// TIA Portal V15.1 export
// export: Created 2024-05-17T05:38:17.1171351Z, ExportSetting WithDefaults, DisplayName Totally Integrated Automation Portal, DisplayVersion V15.1 Update 5, DisplayName TIA Portal Openness, DisplayVersion V15.1 Update 5, DisplayName SINAMICS Startdrive Advanced, DisplayVersion V15.1, DisplayName G130, G150, S120, S150, SINAMICS MV, S210, DisplayVersion V15.1, DisplayName G110M, G120, G120C, G120D, G120P, DisplayVersion V15.1, DisplayName STEP 7 Professional, DisplayVersion V15.1 Update 5, DisplayName STEP 7 Safety, DisplayVersion V15.1, DisplayName WinCC Professional, DisplayVersion V15.1 Update 5, DisplayName SIMATIC Visualization Architect, DisplayVersion V15.1
DATA_BLOCK "_209220ZS01Passiv"   // DB373
{ S7_Optimized_Access := 'FALSE' }
AUTHOR : VCC
VERSION : 0.1
// stored: AutoNumber false, DBAccessibleFromOPCUA true, IsOnlyStoredInLoadMemory false, IsWriteProtectedInAS false
   VAR RETAIN
      AA_209000AK04JX37QF5270 { ExternalAccessible := 'False'; ExternalVisible := 'False'; ExternalWritable := 'False'} : Bool;   // Passivation alarm - ET200sp I/O - Safety Card QF5270
      AA_209000AK04JX37QF5276 { ExternalAccessible := 'False'; ExternalVisible := 'False'; ExternalWritable := 'False'} : Bool;   // Passivation alarm - ET200sp I/O - Safety Card QF5276
      AA_209220AS10JX50IF6000 { ExternalAccessible := 'False'; ExternalVisible := 'False'; ExternalWritable := 'False'} : Bool;   // Passivation alarm - ET200sp I/O - Safety Card IF6000
      AA_209220AX01JX51IF6050 { ExternalAccessible := 'False'; ExternalVisible := 'False'; ExternalWritable := 'False'} : Bool;   // Passivation alarm - ET200sp I/O - Safety Card IF6050
      AA_209220AS11JX52IF6100 { ExternalAccessible := 'False'; ExternalVisible := 'False'; ExternalWritable := 'False'} : Bool;   // Passivation alarm - ET200sp I/O - Safety Card IF6100
      AA_209220AX02JX53IF6150 { ExternalAccessible := 'False'; ExternalVisible := 'False'; ExternalWritable := 'False'} : Bool;   // Passivation alarm - ET200sp I/O - Safety Card IF6150
      AA_209220AS20JX58IF6200 { ExternalAccessible := 'False'; ExternalVisible := 'False'; ExternalWritable := 'False'} : Bool;   // Passivation alarm - ET200sp I/O - Safety Card IF6200
      AA_209000AK04M1UE140 { ExternalAccessible := 'False'; ExternalVisible := 'False'; ExternalWritable := 'False'} : Bool;   // Passivation alarm - MoviDrive - 220CR21M1
      AA_209000AK04M4UE141 { ExternalAccessible := 'False'; ExternalVisible := 'False'; ExternalWritable := 'False'} : Bool;   // Passivation alarm - MoviDrive - 220CS22M4ME1 (Power)
      AA_209000AK04M4UE142 { ExternalAccessible := 'False'; ExternalVisible := 'False'; ExternalWritable := 'False'} : Bool;   // Passivation alarm - MoviDrive - 220CS22M4ME2 (Brake)
      AA_209000AK04M1UE143 { ExternalAccessible := 'False'; ExternalVisible := 'False'; ExternalWritable := 'False'} : Bool;   // Passivation alarm - MoviDrive - 220CR23M1
      AA_209220CHB21M14UE144 { ExternalAccessible := 'False'; ExternalVisible := 'False'; ExternalWritable := 'False'} : Bool;   // Passivation alarm - MoviFit - 220CHB21M14
      "209000AK04JX37QF5270AlarmABCondition" { ExternalAccessible := 'False'; ExternalVisible := 'False'; ExternalWritable := 'False'} : Bool;   // Alarm AB condition
      "209000AK04JX37QF5276AlarmABCondition" { ExternalAccessible := 'False'; ExternalVisible := 'False'; ExternalWritable := 'False'} : Bool;   // Alarm AB condition
      "209220AS10JX50IF6000AlarmABCondition" { ExternalAccessible := 'False'; ExternalVisible := 'False'; ExternalWritable := 'False'} : Bool;   // Alarm AB condition
      "209220AX01JX51IF6050AlarmABCondition" { ExternalAccessible := 'False'; ExternalVisible := 'False'; ExternalWritable := 'False'} : Bool;   // Alarm AB condition
      "209220AS11JX52IF6100AlarmABCondition" { ExternalAccessible := 'False'; ExternalVisible := 'False'; ExternalWritable := 'False'} : Bool;   // Alarm AB condition
      "209220AX02JX53IF6150AlarmABCondition" { ExternalAccessible := 'False'; ExternalVisible := 'False'; ExternalWritable := 'False'} : Bool;   // Alarm AB condition
      "209220AS20JX58IF6200AlarmABCondition" { ExternalAccessible := 'False'; ExternalVisible := 'False'; ExternalWritable := 'False'} : Bool;   // Alarm AB condition
      "209000AK04M1UE140AlarmABCondition" { ExternalAccessible := 'False'; ExternalVisible := 'False'; ExternalWritable := 'False'} : Bool;   // Alarm AB condition
      "209000AK04M4UE141AlarmABCondition" { ExternalAccessible := 'False'; ExternalVisible := 'False'; ExternalWritable := 'False'} : Bool;   // Alarm AB condition
      "209000AK04M4UE142AlarmABCondition" { ExternalAccessible := 'False'; ExternalVisible := 'False'; ExternalWritable := 'False'} : Bool;   // Alarm AB condition
      "209000AK04M1UE143AlarmABCondition" { ExternalAccessible := 'False'; ExternalVisible := 'False'; ExternalWritable := 'False'} : Bool;   // Alarm AB condition
      "209220CHB21M14UE144AlarmABCondition" { ExternalAccessible := 'False'; ExternalVisible := 'False'; ExternalWritable := 'False'} : Bool;   // Alarm AB condition
      H_209000AK04JX37QF5270IAnim : Word;   // HMI Animation of the icon
      H_209000AK04JX37QF5276IAnim : Word;   // HMI Animation of the icon
      H_209220AS10JX50IF6000IAnim : Word;   // HMI Animation of the icon
      H_209220AX01JX51IF6050IAnim : Word;   // HMI Animation of the icon
      H_209220AS11JX52IF6100IAnim : Word;   // HMI Animation of the icon
      H_209220AX02JX53IF6150IAnim : Word;   // HMI Animation of the icon
      H_209220AS20JX58IF6200IAnim : Word;   // HMI Animation of the icon
      H_209000AK04M1UE140IAnim : Word;   // HMI Animation of the icon
      H_209000AK04M4UE141IAnim : Word;   // HMI Animation of the icon
      H_209000AK04M4UE142IAnim : Word;   // HMI Animation of the icon
      H_209000AK04M1UE143IAnim : Word;   // HMI Animation of the icon
      H_209220CHB21M14UE144IAnim : Word;   // HMI Animation of the icon
      H_Anim : Word;   // Animation
      H_DBnr : Int;   // DB number
      AlarmA { ExternalAccessible := 'False'; ExternalVisible := 'False'; ExternalWritable := 'False'} : Bool;   // Summary Alarm A
      AlarmB { ExternalAccessible := 'False'; ExternalVisible := 'False'; ExternalWritable := 'False'} : Bool;   // Summary Alarm B
      AlarmC { ExternalAccessible := 'False'; ExternalVisible := 'False'; ExternalWritable := 'False'} : Bool;   // Summary Alarm C
      AlarmD { ExternalAccessible := 'False'; ExternalVisible := 'False'; ExternalWritable := 'False'} : Bool;   // Summary Alarm D
      AlarmABCondition { ExternalAccessible := 'False'; ExternalVisible := 'False'; ExternalWritable := 'False'} : Bool;   // Alarm AB Condition
      PassivationError { ExternalAccessible := 'False'; ExternalVisible := 'False'; ExternalWritable := 'False'} : Bool;   // There is one ore more Passivation Errors active
      FeedBackError { ExternalAccessible := 'False'; ExternalVisible := 'False'; ExternalWritable := 'False'} : Bool;   // There is one ore more FeedBack Errors active
      "AckReqSendRcvDP/PN" { ExternalAccessible := 'False'; ExternalVisible := 'False'; ExternalWritable := 'False'} : Bool;   // Ack.Req from DP/DP or PN/PN couplers
   END_VAR
BEGIN
END_DATA_BLOCK
